// TIA Portal V21 export
DATA_BLOCK "CipPulse"   // DB204
{ S7_Optimized_Access := 'FALSE' }
// stored: AutoNumber false
   VAR
      RE : Array[0..25] of Bool;
      D500EventsTimer : Array[0..25] of IEC_TIMER;
   END_VAR
BEGIN
END_DATA_BLOCK
